// TIA Portal project "hmı_modülü_baharat_karıştırıcı" (V17)

(* hardware
DEVICE "S7-1200 station_1"  S7-1200 Station
   slot 0: "Rack_0"  S7-1200 Rack  Rack  V1.0
   slot 1: "PLC_1"  CPU 1214C DC/DC/DC  6ES7 214-1AG40-0XB0  V4.5
DEVICE "HMI_1"  KTP900 Basic PN
   slot 0: "HMI_1"  KTP900 Basic PN  6AV2 123-2JB03-0AX0  17.0.0.0
   slot 1: "HMI_RT_1"  KTP900 Basic PN  6AV2 123-2JB03-0AX0  17.0.0.0
   slot 5: "HMI_1.IE_CP_1"  PROFINET Interface  17.0.0.0
      slot 1: "PROFINET Interface_1"  PROFINET Interface
         slot 1: "Port_1"  Port
*)

// ===== PLC "PLC_1"  CPU 1214C DC/DC/DC =====

VAR_GLOBAL   // PLC tag table "Default tag table"
   "System_Byte" AT %MB1 : Byte;
   "FirstScan" AT %M1.0 : Bool;
   "DiagStatusUpdate" AT %M1.1 : Bool;
   "AlwaysTRUE" AT %M1.2 : Bool;
   "AlwaysFALSE" AT %M1.3 : Bool;
   "Clock_Byte" AT %MB0 : Byte;
   "Clock_10Hz" AT %M0.0 : Bool;
   "Clock_5Hz" AT %M0.1 : Bool;
   "Clock_2.5Hz" AT %M0.2 : Bool;
   "Clock_2Hz" AT %M0.3 : Bool;
   "Clock_1.25Hz" AT %M0.4 : Bool;
   "Clock_1Hz" AT %M0.5 : Bool;
   "Clock_0.625Hz" AT %M0.6 : Bool;
   "Clock_0.5Hz" AT %M0.7 : Bool;
   "stop" AT %I0.0 : Bool;
   "start" AT %I0.1 : Bool;
   "sistem" AT %M20.0 : Bool;
   "termik" AT %I0.2 : Bool;
   "motor yön 1" AT %Q0.0 : Bool;
   "motor yön 2" AT %Q0.1 : Bool;
   "lamba yön 1" AT %Q0.2 : Bool;
   "lamba yön 2" AT %Q0.3 : Bool;
   "lamba arıza" AT %Q0.6 : Bool;
   "termostat" AT %I0.3 : Bool;
   "ısıtıcı" AT %Q0.4 : Bool;
   "lamba ısıtıcı" AT %Q0.5 : Bool;
   "Tag_1" AT %Q0.7 : Bool;
   "Tag_2" AT %Q1.0 : Bool;
   "Tag_3" AT %MW500 : Int;
   "Tag_4" AT %MW50 : Word;
   "Tag_5" AT %MW5000 : Word;
   "Tag_6" AT %MW51 : Word;
   "Tag_7" AT %MW5001 : Word;
END_VAR

// folder: System blocks/Program resources

DATA_BLOCK "yön 1 çalışma zaman"   // DB1
{ S7_Optimized_Access := 'TRUE' }
AUTHOR : Simatic
FAMILY : IEC
NAME : IEC_TMR
VERSION : 1.0
// stored: InstanceOfName IEC_TIMER
"IEC_TIMER"
BEGIN
END_DATA_BLOCK

DATA_BLOCK "sayıcı"   // DB2
{ S7_Optimized_Access := 'TRUE' }
AUTHOR : Simatic
FAMILY : IEC
NAME : CNTR
VERSION : 1.0
// stored: InstanceOfName IEC_COUNTER
"IEC_COUNTER"
BEGIN
END_DATA_BLOCK

DATA_BLOCK "yön1 bekleme zaman"   // DB6
{ S7_Optimized_Access := 'TRUE' }
AUTHOR : Simatic
FAMILY : IEC
NAME : IEC_TMR
VERSION : 1.0
// stored: InstanceOfName IEC_TIMER
"IEC_TIMER"
BEGIN
END_DATA_BLOCK

DATA_BLOCK "yön 2 çalışma zaman"   // DB7
{ S7_Optimized_Access := 'TRUE' }
AUTHOR : Simatic
FAMILY : IEC
NAME : IEC_TMR
VERSION : 1.0
// stored: InstanceOfName IEC_TIMER
"IEC_TIMER"
BEGIN
END_DATA_BLOCK

DATA_BLOCK "yön 2 bekleme zaman"   // DB8
{ S7_Optimized_Access := 'TRUE' }
AUTHOR : Simatic
FAMILY : IEC
NAME : IEC_TMR
VERSION : 1.0
// stored: InstanceOfName IEC_TIMER
"IEC_TIMER"
BEGIN
END_DATA_BLOCK

// folder: (top level)

FUNCTION "Block_1" : Void   // FC1, LAD
{ S7_Optimized_Access := 'FALSE' }
VERSION : 0.1
   VAR_INPUT
      start : Bool;
      stop : Bool;
      termik : Bool;
   END_VAR
   VAR_OUTPUT
      "lamba ısıtıcı" : Bool;
      "lamba arıza" : Bool;
      "lamba yön 2" : Bool;
      "lamba yön 1" : Bool;
   END_VAR
   VAR_TEMP   // added for the SCL form of the ladder/FBD networks
      _w1 : Bool;
      _w2 : Bool;
   END_VAR
BEGIN

REGION Network 1
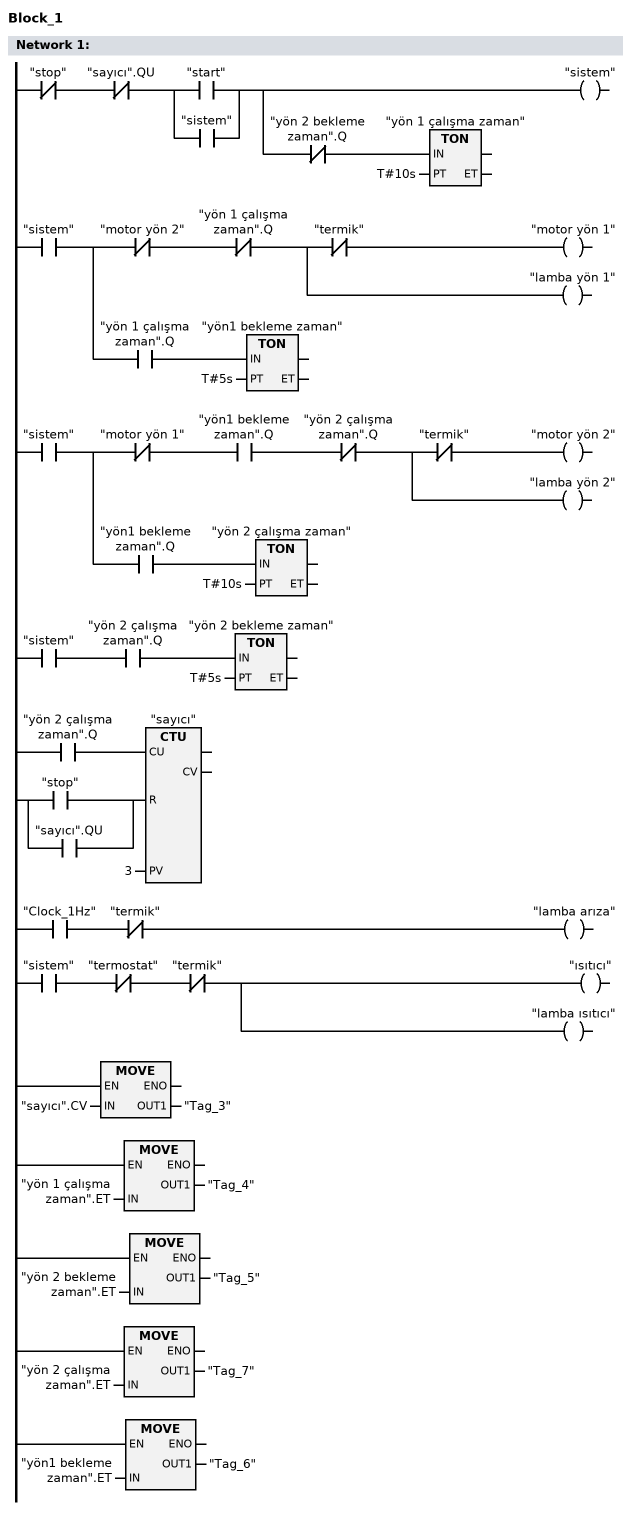
   "sistem" := NOT "stop" AND NOT "sayıcı".QU AND ("start" OR "sistem");
   "yön 1 çalışma zaman".TON(IN := "sistem" AND NOT "yön 2 bekleme zaman".Q, PT := T#10s);
   #_w1 := "sistem" AND NOT "motor yön 2" AND NOT "yön 1 çalışma zaman".Q;
   "motor yön 1" := #_w1 AND NOT "termik";
   "lamba yön 1" := #_w1;
   "yön1 bekleme zaman".TON(IN := "sistem" AND "yön 1 çalışma zaman".Q, PT := T#5s);
   #_w2 := "sistem" AND NOT "motor yön 1" AND "yön1 bekleme zaman".Q AND NOT "yön 2 çalışma zaman".Q;
   "motor yön 2" := #_w2 AND NOT "termik";
   "lamba yön 2" := #_w2;
   "yön 2 çalışma zaman".TON(IN := "sistem" AND "yön1 bekleme zaman".Q, PT := T#10s);
   "yön 2 bekleme zaman".TON(IN := "sistem" AND "yön 2 çalışma zaman".Q, PT := T#5s);
   "sayıcı".CTU(CU := "yön 2 çalışma zaman".Q, R := "stop" OR "sayıcı".QU, PV := 3);
   "lamba arıza" := "Clock_1Hz" AND NOT "termik";
   "ısıtıcı" := "sistem" AND NOT "termostat" AND NOT "termik";
   "lamba ısıtıcı" := "ısıtıcı";
   "Tag_3" := "sayıcı".CV;
   "Tag_4" := "yön 1 çalışma zaman".ET;
   "Tag_5" := "yön 2 bekleme zaman".ET;
   "Tag_7" := "yön 2 çalışma zaman".ET;
   "Tag_6" := "yön1 bekleme zaman".ET;
END_REGION
END_FUNCTION

FUNCTION "Block_2" : Void   // FC2, LAD
{ S7_Optimized_Access := 'TRUE' }
VERSION : 0.1
BEGIN

REGION Network 1
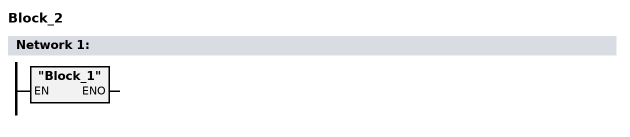
   RUNG wire#powerrail
      "Block_1"()
   END_RUNG
   // the same network as SCL:
   "Block_1"();
END_REGION
END_FUNCTION

ORGANIZATION_BLOCK "Main"   // OB1, LAD, ProgramCycle
TITLE = "Main Program Sweep (Cycle)"
{ S7_Optimized_Access := 'TRUE' }
VERSION : 0.1
   VAR_INPUT
      Initial_Call : Bool;   // Initial call of this OB
      Remanence : Bool;   // =True, if remanent data are available
   END_VAR
BEGIN

REGION Network 1
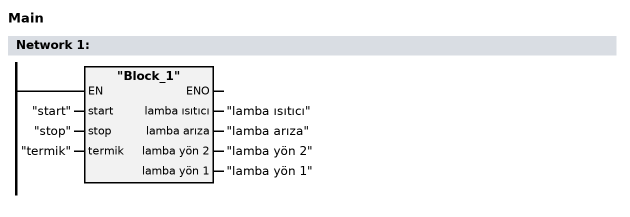
   RUNG wire#powerrail
      "Block_1"(start := "start", stop := "stop", termik := "termik", "lamba ısıtıcı" => "lamba ısıtıcı", "lamba arıza" => "lamba arıza", "lamba yön 2" => "lamba yön 2", "lamba yön 1" => "lamba yön 1")
   END_RUNG
   // the same network as SCL:
   "Block_1"(start := "start",
             stop := "stop",
             termik := "termik",
             "lamba ısıtıcı" => "lamba ısıtıcı",
             "lamba arıza" => "lamba arıza",
             "lamba yön 2" => "lamba yön 2",
             "lamba yön 1" => "lamba yön 1");
END_REGION
END_ORGANIZATION_BLOCK

(* ===== HMI "HMI_RT_1" =====
system functions are stored by id; their names below are inferred from use
connection "HMI_Connection_1": ETHERNET, SMART_S7_1200_OMS

HMI tags "Default tag table"
   "start" : Bool = PLC start AT %I0.1, 1 s
   "stop" : Bool = PLC stop AT %I0.0, 1 s
   "sistem" : Bool = PLC sistem AT %M20.0, 1 s
   "termik" : Bool = PLC termik AT %I0.2, 1 s
   "motor yön 1" : Bool = PLC "motor yön 1" AT %Q0.0, 1 s
   "motor yön 2" : Bool = PLC "motor yön 2" AT %Q0.1, 1 s
   "lamba yön1" : Bool = PLC "lamba yön 1" AT %Q0.2, 1 s
   "lamba yön2" : Bool = PLC "lamba yön 2" AT %Q0.3, 1 s
   "ısıtıcı" : Bool = PLC ısıtıcı AT %Q0.4, 1 s
   "arıza" : Bool = PLC "lamba arıza" AT %Q0.6, 1 s
   "sayıcı_değerş" : Int = PLC Tag_3 AT %MW500, 1 s
   "çalışma 1" : Word = PLC Tag_4 AT %MW50, 1 s
   "çalışma 2" : Word = PLC Tag_5 AT %MW5000, 1 s
   "bekleme 2" : Word = PLC Tag_7 AT %MW5001, 1 s
   "bekleme 1" : Word = PLC Tag_6 AT %MW51, 1 s

Template "Template_1" 800x480
   Button "Exit" at 722,440 size 55x39; TextOff 'Exit'; PictureOff "ExitRuntime_KTP900_Basic_PN_TR"; PictureOn "ExitRuntime_KTP900_Basic_PN_TR"
      on Release: StopRuntime(0)
   Button "Template_Button" at 622,440 size 55x39; TextOff 'Text'
   Button "Template_Button_1" at 522,440 size 55x39; TextOff 'Text'
   Button "Template_Button_2" at 422,440 size 55x39; TextOff 'Text'
   Button "Template_Button_3" at 322,440 size 55x39; TextOff 'Text'
   Button "Template_Button_4" at 222,440 size 55x39; TextOff 'Text'
   Button "Alarms" at 122,440 size 55x39; TextOff 'Alarms'; PictureOff "AlarmDisplay_KTP900_Basic_PN_TR"; PictureOn "AlarmDisplay_KTP900_Basic_PN_TR"
      on Release: function_ef3f5d25("Alarm window_Unacknowledged", -1)
   Button "Start screen" at 22,440 size 55x39; TextOff 'Start screen'; PictureOff "NavigateHome_KTP900_Basic_PN_TR"; PictureOn "NavigateHome_KTP900_Basic_PN_TR"
      on Release: ActivateScreen("Root screen", 0)
   DateTimeField "HmiScreenItemData" at 695,20 size 105x20
   DateTimeField "HmiScreenItemData_1" at 695,0 size 105x20
   GraphicView "Logo" at 0,0 size 71x40; Picture "Logo of HMI_1"

screen "Root screen" 800x480, template "Template_1"
   on GenerateScreen: SetTag("start", 1)
   TextField "HmiScreenItemData" at 79,288 size 640x22; Text 'HMI ALİ EDİTİON'
   Button "Button_1" at 197,98 size 132x40; TextOff 'START'
      on Press: SetBit("start")
   Button "Button_2" at 483,97 size 138x41; TextOff 'STOP'
      on Press: SetBit("stop")
   GraphicIOField "PlotLight_Round_G" at 29,344 size 95x72; PictureOn "PilotLight_Round_G_On_256c"; PictureOff "PilotLight_Round_G_Off_256c"
      ProcessValue <- "lamba yön1"
   GraphicIOField "PlotLight_Round_R" at 172,343 size 93x76; PictureOn "PilotLight_Round_R_On_256c"; PictureOff "PilotLight_Round_R_Off_256c"
      ProcessValue <- "lamba yön2"
   GraphicIOField "PlotLight_Square_G" at 317,196 size 84x66; PictureOn "PilotLight_Square_G_On_256c"; PictureOff "PilotLight_Square_G_Off_256c"
      ProcessValue <- "termik"
   GraphicIOField "PlotLight_Square_R" at 462,196 size 76x65; PictureOn "PilotLight_Square_R_On_256c"; PictureOff "PilotLight_Square_R_Off_256c"
      ProcessValue <- "ısıtıcı"
   TextField "Text field_1" at 51,140 size 76x40; Text 'İLERİ YÖN'
   TextField "Text field_2" at 171,158 size 73x22; Text 'GERİ YÖN'
   TextField "Text field_3" at 323,158 size 58x22; Text 'TERMİK'
   TextField "Text field_4" at 473,160 size 55x22; Text 'ISITICI'
   GraphicIOField "PlotLight_Square_N_Mono" at 581,195 size 75x68; PictureOn "PilotLight_Square_N_On_mono"; PictureOff "PilotLight_Square_N_Off_mono"
      ProcessValue <- "sistem"
   GraphicIOField "PlotLight_Square_GN" at 683,198 size 79x66; PictureOn "PilotLight_Square_GN_On_256c"; PictureOff "PilotLight_Square_GN_Off_256c"
      ProcessValue <- "arıza"
   TextField "Text field_5" at 586,162 size 56x22; Text 'SİSTEM'
   TextField "Text field_6" at 696,158 size 45x22; Text 'ARIZA'
   IOField "I/O field_1" at 363,384 size 112x32; FormatPattern s9
      ProcessValue <- "sayıcı_değerş"
   IOField "I/O field_2" at 51,229 size 55x32; FormatPattern 999999
      ProcessValue <- "çalışma 1"
   IOField "I/O field_3" at 51,300 size 52x32; FormatPattern 999999
      ProcessValue <- "bekleme 1"
   IOField "I/O field_5" at 188,229 size 56x32; FormatPattern 999999
      ProcessValue <- "bekleme 2"
   TextField "Text field_7" at 374,343 size 85x22; Text 'TUR SAYISI'
   TextField "Text field_8" at 17,195 size 118x22; Text 'ÇALIŞMA SÜRESİ'
   TextField "Text field_9" at 149,195 size 118x22; Text 'ÇALIŞMA SÜRESİ'
   TextField "Text field_10" at 17,272 size 119x22; Text 'BEKLEME SÜRESİ'
   TextField "Text field_11" at 149,272 size 119x22; Text 'BEKLEME SÜRESİ'
   TextField "Text field_12" at 172,310 size 13x22; Text 'Text'
   IOField "I/O field_6" at 184,300 size 53x32; FormatPattern 999999
      ProcessValue <- "çalışma 2"
*)